Universal Robots PolyScope program: mambo.urp

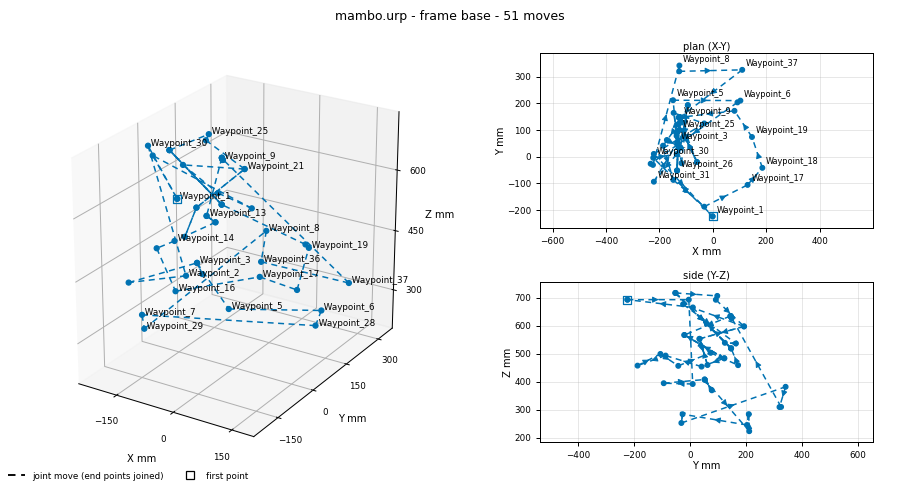
[picture p0: tool path of mambo.urp in frame base, 51 of 51 moves have a stored position in this frame; points joined in program order, loops and branches not executed]
Program mambo (installation=schmalz directory=/programs createdIn=5.3.0.64176 lastSavedIn=5.3.0.64176 robotSerialNumber=20185300040)
Calibrated DH parameters: a=[0, -0.24355, -0.2132, 0, 0, 0]; d=[0.15185, 0, 0, 0.13105, 0.08535, 0.0921]; alpha=[1.570796, 0, 0, 1.570796, -1.570796, 0]; deltaTheta=[0, 0, 0, 0, 0, 0]
Robot Program (runOnlyOnce=false)
  'posicio inici'
  MoveJ speed 150 deg/s, acceleration 150 deg/s^2 (useActiveTCP=true) feature=Base
    Waypoint Waypoint_1: TCP in base x=-0.824 y=-223.149 z=693.949 mm, rx=-0.0017 ry=-2.2201 rz=2.22 rad; joints [-0.035, -89.919, -0.062, -89.93, -0.088, -0.125] deg
  Wait Sleep waitTime=1
  MoveJ speed 60 deg/s, acceleration 80 deg/s^2 (useActiveTCP=true) feature=Base
    Waypoint Waypoint_30: TCP in base x=-223.116 y=-3.912 z=693.95 mm, rx=-1.2004 ry=-1.2209 rz=1.2177 rad; joints [-89.059, -90.033, -0.04, -89.953, -0.124, -0.127] deg
  Wait Sleep waitTime=1.6
  'move down'
  MoveJ speed 150 deg/s, acceleration 150 deg/s^2 (useActiveTCP=true) feature=Base
    Waypoint Waypoint_2: TCP in base x=-135.234 y=10.106 z=392.808 mm, rx=-1.5933 ry=-0.0499 rz=0.0467 rad; joints [-88.964, -175.644, 134.862, -137.895, -87.524, -0.132] deg
  'move around'
  MoveJ speed 360 deg/s, acceleration 360 deg/s^2 (useActiveTCP=true) feature=Base
    Waypoint Waypoint_31: TCP in base x=-220.784 y=-93.368 z=395.621 mm, rx=-1.1585 ry=-1.2927 rz=1.3141 rad; joints [-88.833, -175.384, 134.818, -138.339, 6.036, -0.153] deg
  'cap avall'
  MoveJ speed 360 deg/s, acceleration 360 deg/s^2 (useActiveTCP=true) feature=Base
    Waypoint Waypoint_3: TCP in base x=-133.135 y=52.728 z=408.846 mm, rx=-1.5319 ry=-0.1392 rz=-0.0523 rad; joints [-84.379, -156.87, 136.847, -161.86, -92.314, -7.153] deg
  MoveJ speed 360 deg/s, acceleration 360 deg/s^2 (useActiveTCP=true) feature=Base
    Waypoint Waypoint_4: TCP in base x=-135.698 y=78.393 z=370.338 mm, rx=-1.896 ry=-0.1853 rz=-0.0565 rad; joints [-84.353, -156.912, 137.023, -140.966, -92.318, -7.163] deg
  'cap amunt'
  MoveJ speed 360 deg/s, acceleration 360 deg/s^2 (useActiveTCP=true) feature=Base
    Waypoint Waypoint_3: TCP in base x=-133.135 y=52.728 z=408.846 mm, rx=-1.5319 ry=-0.1392 rz=-0.0523 rad; joints [-84.379, -156.87, 136.847, -161.86, -92.314, -7.153] deg
  'hand on the ground'
  MoveJ speed 360 deg/s, acceleration 360 deg/s^2 (useActiveTCP=true) feature=Base
    Waypoint Waypoint_5: TCP in base x=-148.892 y=211.875 z=224.279 mm, rx=-2.7527 ry=-0.2984 rz=-0.0629 rad; joints [-84.355, -107.408, 137.019, -140.967, -92.316, -7.165] deg
  'step left'
  MoveJ speed 360 deg/s, acceleration 360 deg/s^2 (useActiveTCP=true) feature=Base
    Waypoint Waypoint_6: TCP in base x=103.306 y=210.335 z=285.176 mm, rx=-2.2966 ry=1.1384 rz=-0.5195 rad; joints [-149.105, -123.568, 136.822, -140.905, -92.243, -7.137] deg
  MoveJ speed 360 deg/s, acceleration 360 deg/s^2 (useActiveTCP=true) feature=Base
    Waypoint Waypoint_28: TCP in base x=92.285 y=203.712 z=246.45 mm, rx=-2.5753 ry=1.2658 rz=-0.3089 rad; joints [-149.112, -123.457, 136.825, -122.33, -92.244, -7.137] deg
  'step right'
  MoveJ speed 360 deg/s, acceleration 360 deg/s^2 (useActiveTCP=true) feature=Base
    Waypoint Waypoint_7: TCP in base x=-232.811 y=-26.127 z=284.929 mm, rx=-2.0676 ry=-1.4429 rz=0.3615 rad; joints [-26.553, -123.575, 136.866, -140.898, -92.245, -7.137] deg
  MoveJ speed 360 deg/s, acceleration 360 deg/s^2 (useActiveTCP=true) feature=Base
    Waypoint Waypoint_29: TCP in base x=-224.234 y=-30.449 z=253.639 mm, rx=-2.2651 ry=-1.5899 rz=0.2136 rad; joints [-26.545, -123.574, 136.867, -125.919, -92.241, -7.122] deg
  'step front'
  MoveJ speed 360 deg/s, acceleration 360 deg/s^2 (useActiveTCP=true) feature=Base
    Waypoint Waypoint_8: TCP in base x=-125.24 y=341.779 z=382.876 mm, rx=-2.4947 ry=-0.1311 rz=-0.1034 rad; joints [-90.371, -88.956, 86.351, -124.378, -92.24, -7.138] deg
  MoveJ speed 360 deg/s, acceleration 360 deg/s^2 (useActiveTCP=true) feature=Base
    Waypoint Waypoint_36: TCP in base x=-125.934 y=320.003 z=310.577 mm, rx=-2.9382 ry=-0.1696 rz=-0.0744 rad; joints [-90.296, -88.943, 92.058, -104.601, -92.155, -7.119] deg
  'step side'
  MoveJ speed 360 deg/s, acceleration 360 deg/s^2 (useActiveTCP=true) feature=Base
    Waypoint Waypoint_37: TCP in base x=110.144 y=325.613 z=310.939 mm, rx=-2.8414 ry=0.8568 rz=-0.1736 rad; joints [-130.459, -88.994, 92.044, -104.599, -92.217, -7.122] deg
  MoveJ speed 130 deg/s, acceleration 130 deg/s^2 (useActiveTCP=true) feature=Base
    Waypoint Waypoint_9: TCP in base x=-124.361 y=147.084 z=632.656 mm, rx=-1.782 ry=-0.0641 rz=-0.1388 rad; joints [-91.291, -107.109, 47.563, -108.401, -92.12, -7.127] deg
  Wait NoWait
  'clap once'
  MoveJ speed 150 deg/s, acceleration 150 deg/s^2 (useActiveTCP=true) feature=Base
    Waypoint Waypoint_10: TCP in base x=-124.49 y=149.03 z=629.258 mm, rx=-1.8133 ry=-0.0671 rz=-0.1366 rad; joints [-91.243, -107.089, 47.543, -106.599, -92.088, -7.12] deg
  MoveJ speed 150 deg/s, acceleration 150 deg/s^2 (useActiveTCP=true) feature=Base
    Waypoint Waypoint_11: TCP in base x=-124.409 y=145.217 z=635.714 mm, rx=-1.7534 ry=-0.0624 rz=-0.1396 rad; joints [-91.287, -107.105, 47.563, -110.044, -92.122, -7.129] deg
  Wait Sleep waitTime=0.6
  'clap twice'
  MoveJ speed 150 deg/s, acceleration 150 deg/s^2 (useActiveTCP=true) feature=Base
    Waypoint Waypoint_10: TCP in base x=-124.49 y=149.03 z=629.258 mm, rx=-1.8133 ry=-0.0671 rz=-0.1366 rad; joints [-91.243, -107.089, 47.543, -106.599, -92.088, -7.12] deg
  MoveJ speed 150 deg/s, acceleration 150 deg/s^2 (useActiveTCP=true) feature=Base
    Waypoint Waypoint_11: TCP in base x=-124.409 y=145.217 z=635.714 mm, rx=-1.7534 ry=-0.0624 rz=-0.1396 rad; joints [-91.287, -107.105, 47.563, -110.044, -92.122, -7.129] deg
  MoveJ speed 150 deg/s, acceleration 150 deg/s^2 (useActiveTCP=true) feature=Base
    Waypoint Waypoint_10: TCP in base x=-124.49 y=149.03 z=629.258 mm, rx=-1.8133 ry=-0.0671 rz=-0.1366 rad; joints [-91.243, -107.089, 47.543, -106.599, -92.088, -7.12] deg
  MoveJ speed 150 deg/s, acceleration 150 deg/s^2 (useActiveTCP=true) feature=Base
    Waypoint Waypoint_11: TCP in base x=-124.409 y=145.217 z=635.714 mm, rx=-1.7534 ry=-0.0624 rz=-0.1396 rad; joints [-91.287, -107.105, 47.563, -110.044, -92.122, -7.129] deg
  'estribillu mode 1'
  MoveJ speed 150 deg/s, acceleration 150 deg/s^2 (useActiveTCP=true) feature=Base
    Waypoint Waypoint_13: TCP in base x=-59.578 y=-19.761 z=567.729 mm, rx=-1.6686 ry=0.7159 rz=-1.0662 rad; joints [-99.242, -141.569, 77.085, -103.183, -144.973, -8.251] deg
  MoveJ speed 150 deg/s, acceleration 150 deg/s^2 (useActiveTCP=true) feature=Base
    Waypoint Waypoint_12: TCP in base x=-127.936 y=122.86 z=484.642 mm, rx=-1.6109 ry=-0.0779 rz=-0.1183 rad; joints [-91.017, -33.433, -113.259, -30.974, -90.593, -7.127] deg
  MoveJ speed 150 deg/s, acceleration 150 deg/s^2 (useActiveTCP=true) feature=Base
    Waypoint Waypoint_13: TCP in base x=-59.578 y=-19.761 z=567.729 mm, rx=-1.6686 ry=0.7159 rz=-1.0662 rad; joints [-99.242, -141.569, 77.085, -103.183, -144.973, -8.251] deg
  MoveJ speed 150 deg/s, acceleration 150 deg/s^2 (useActiveTCP=true) feature=Base
    Waypoint Waypoint_12: TCP in base x=-127.936 y=122.86 z=484.642 mm, rx=-1.6109 ry=-0.0779 rz=-0.1183 rad; joints [-91.017, -33.433, -113.259, -30.974, -90.593, -7.127] deg
  'estribillu mode 2'
  MoveJ speed 150 deg/s, acceleration 150 deg/s^2 (useActiveTCP=true) feature=Base
    Waypoint Waypoint_14: motionParameters(blendRadius=0.05); TCP in base x=-186.309 y=41.586 z=454.903 mm, rx=-1.7872 ry=-0.6708 rz=0.3146 rad; joints [-55.578, -33.494, -113.137, -14.702, -90.543, -7.116] deg
  MoveJ speed 150 deg/s, acceleration 150 deg/s^2 (useActiveTCP=true) feature=Base
    Waypoint Waypoint_15: motionParameters(blendRadius=0.05); TCP in base x=-147.873 y=-86.71 z=494.359 mm, rx=-1.2266 ry=-0.9847 rz=0.8802 rad; joints [-19.024, -33.468, -113.195, -36.982, -90.544, -7.118] deg
  MoveJ speed 150 deg/s, acceleration 150 deg/s^2 (useActiveTCP=true) feature=Base
    Waypoint Waypoint_16: motionParameters(blendRadius=0.05); TCP in base x=-32.144 y=-186.918 z=458.41 mm, rx=-0.9509 ry=-1.9368 rz=1.4208 rad; joints [36.9, -33.462, -113.189, -16.538, -90.544, -1.207] deg
  MoveJ speed 120 deg/s, acceleration 120 deg/s^2 (useActiveTCP=true) feature=Base
    Waypoint Waypoint_17: motionParameters(blendRadius=0.044); TCP in base x=130.235 y=-105.29 z=500.108 mm, rx=-0.0064 ry=-2.0638 rz=2.3575 rad; joints [89.894, -33.467, -113.196, -40.94, -90.386, -0.193] deg
  MoveJ speed 150 deg/s, acceleration 150 deg/s^2 (useActiveTCP=true) feature=Base
    Waypoint Waypoint_18: motionParameters(blendRadius=0.05); TCP in base x=185.501 y=-41.46 z=457.651 mm, rx=-0.8139 ry=2.1842 rz=-1.6731 rad; joints [124.08, -33.465, -113.191, -16.151, -90.399, -7.089] deg
  MoveJ speed 150 deg/s, acceleration 150 deg/s^2 (useActiveTCP=true) feature=Base
    Waypoint Waypoint_19: motionParameters(blendRadius=0.05); TCP in base x=146.639 y=74.125 z=504.117 mm, rx=-0.9528 ry=1.3379 rz=-1.7388 rad; joints [154.283, -33.466, -113.194, -43.903, -90.396, -7.109] deg
  MoveJ speed 150 deg/s, acceleration 150 deg/s^2 (useActiveTCP=true) feature=Base
    Waypoint Waypoint_20: motionParameters(blendRadius=0.05); TCP in base x=81.114 y=172.065 z=460.079 mm, rx=-1.6759 ry=0.9998 rz=-0.9017 rad; joints [200.887, -33.455, -113.19, -17.397, -89.51, -7.105] deg
  'estribillu mode 3'
  MoveJ speed 150 deg/s, acceleration 150 deg/s^2 (useActiveTCP=true) feature=Base
    Waypoint Waypoint_22: motionParameters(blendRadius=0); TCP in base x=-126.514 y=147.162 z=519.996 mm, rx=-1.9842 ry=-0.0921 rz=-0.0954 rad; joints [267.883, -45.32, -88.466, -22.477, -89.493, -7.101] deg
  MoveJ speed 150 deg/s, acceleration 150 deg/s^2 (useActiveTCP=true) feature=Base
    Waypoint Waypoint_26: motionParameters(blendRadius=0.05); TCP in base x=-133.87 y=-51.593 z=717.983 mm, rx=-0.8271 ry=-0.0444 rz=-0.1478 rad; joints [267.884, -86.921, -25.009, -110.661, -89.488, -7.099] deg
  MoveJ speed 150 deg/s, acceleration 150 deg/s^2 (useActiveTCP=true) feature=Base
    Waypoint Waypoint_22: motionParameters(blendRadius=0); TCP in base x=-126.514 y=147.162 z=519.996 mm, rx=-1.9842 ry=-0.0921 rz=-0.0954 rad; joints [267.883, -45.32, -88.466, -22.477, -89.493, -7.101] deg
  MoveJ speed 150 deg/s, acceleration 150 deg/s^2 (useActiveTCP=true) feature=Base
    Waypoint Waypoint_26: motionParameters(blendRadius=0.05); TCP in base x=-133.87 y=-51.593 z=717.983 mm, rx=-0.8271 ry=-0.0444 rz=-0.1478 rad; joints [267.884, -86.921, -25.009, -110.661, -89.488, -7.099] deg
  MoveJ speed 150 deg/s, acceleration 150 deg/s^2 (useActiveTCP=true) feature=Base
    Waypoint Waypoint_22: motionParameters(blendRadius=0); TCP in base x=-126.514 y=147.162 z=519.996 mm, rx=-1.9842 ry=-0.0921 rz=-0.0954 rad; joints [267.883, -45.32, -88.466, -22.477, -89.493, -7.101] deg
  MoveJ speed 150 deg/s, acceleration 150 deg/s^2 (useActiveTCP=true) feature=Base
    Waypoint Waypoint_26: motionParameters(blendRadius=0.05); TCP in base x=-133.87 y=-51.593 z=717.983 mm, rx=-0.8271 ry=-0.0444 rz=-0.1478 rad; joints [267.884, -86.921, -25.009, -110.661, -89.488, -7.099] deg
  MoveJ speed 150 deg/s, acceleration 150 deg/s^2 (useActiveTCP=true) feature=Base
    Waypoint Waypoint_25: motionParameters(blendRadius=0.014); TCP in base x=-128.362 y=97.775 z=707.429 mm, rx=-1.382 ry=-0.0677 rz=-0.1281 rad; joints [267.89, -82.809, -10.415, -97.565, -89.487, -7.1] deg
  'fi estribillu'
  MoveJ speed 150 deg/s, acceleration 150 deg/s^2 (useActiveTCP=true) feature=Base
    Waypoint Waypoint_23: TCP in base x=-132.936 y=92.662 z=693.638 mm, rx=-1.5741 ry=-0.0178 rz=0.0144 rad; joints [-90.243, -90.107, 0.158, -89.858, -88.583, -0.125] deg
  'inici trompetes'
  Loop Counting (count=3) loopVariable(name=Loop_1)
    MoveJ speed 360 deg/s, acceleration 360 deg/s^2 (useActiveTCP=true) feature=Base
      Waypoint Waypoint_21: TCP in base x=-93.62 y=193.187 z=598.504 mm, rx=-1.6092 ry=0.0181 rz=0.0116 rad; joints [-118.764, -117.573, 73.22, -133.137, -61.475, -0.126] deg
    MoveJ speed 360 deg/s, acceleration 360 deg/s^2 (useActiveTCP=true) feature=Base
      Waypoint Waypoint_24: TCP in base x=-121.507 y=34.416 z=554.148 mm, rx=-1.6234 ry=-0.0522 rz=0.0123 rad; joints [-65.364, -132.876, 90.562, -134.38, -112.301, -0.129] deg
    MoveJ speed 360 deg/s, acceleration 360 deg/s^2 (useActiveTCP=true) feature=Base
      Waypoint Waypoint_27: TCP in base x=-172.118 y=62.873 z=460.667 mm, rx=-1.5663 ry=-0.025 rz=0.0173 rad; joints [-120.652, -167.743, 114.251, -126.801, -57.803, -0.127] deg
    MoveJ speed 360 deg/s, acceleration 360 deg/s^2 (useActiveTCP=true) feature=Base
      Waypoint Waypoint_24: TCP in base x=-121.507 y=34.416 z=554.148 mm, rx=-1.6234 ry=-0.0522 rz=0.0123 rad; joints [-65.364, -132.876, 90.562, -134.38, -112.301, -0.129] deg
    MoveJ speed 360 deg/s, acceleration 360 deg/s^2 (useActiveTCP=true) feature=Base
      Waypoint Waypoint_21: TCP in base x=-93.62 y=193.187 z=598.504 mm, rx=-1.6092 ry=0.0181 rz=0.0116 rad; joints [-118.764, -117.573, 73.22, -133.137, -61.475, -0.126] deg
  'trompetero'
  Loop Counting (count=4) loopVariable(name=Loop_2)
    MoveJ speed 360 deg/s, acceleration 360 deg/s^2 (useActiveTCP=true) feature=Base
      Waypoint Waypoint_32: TCP in base x=-117.273 y=-24.208 z=677.605 mm, rx=-0.4321 ry=0.5657 rz=-0.6065 rad; joints [-118.678, -120.382, 50.679, -168.263, -115.59, -0.126] deg
    MoveJ speed 360 deg/s, acceleration 360 deg/s^2 (useActiveTCP=true) feature=Base
      Waypoint Waypoint_33: TCP in base x=-146.706 y=164.413 z=537.566 mm, rx=-2.1339 ry=-0.3305 rz=0.7084 rad; joints [-118.359, -123.183, 63.764, -60.885, -34.232, -29.66] deg
    MoveJ speed 360 deg/s, acceleration 360 deg/s^2 (useActiveTCP=true) feature=Base
      Waypoint Waypoint_34: TCP in base x=-32.166 y=124.874 z=539.926 mm, rx=-2.5043 ry=0.2254 rz=-1.0388 rad; joints [-118.379, -123.035, 63.947, -74.975, -118.112, -29.665] deg
    MoveJ speed 360 deg/s, acceleration 360 deg/s^2 (useActiveTCP=true) feature=Base
      Waypoint Waypoint_35: TCP in base x=-220.993 y=10.655 z=666.213 mm, rx=-0.655 ry=-0.8177 rz=-0.6185 rad; joints [-118.37, -121.581, 47.497, -156.348, -41.981, -28.828] deg
    MoveJ speed 150 deg/s, acceleration 150 deg/s^2 (useActiveTCP=true) feature=Base
      Waypoint Waypoint_1: TCP in base x=-0.824 y=-223.149 z=693.949 mm, rx=-0.0017 ry=-2.2201 rz=2.22 rad; joints [-0.035, -89.919, -0.062, -89.93, -0.088, -0.125] deg
